Staubli VAL3: Deplacement.pgx

program Deplacement()
begin
  movej(jInit, flange, mNomSpeed)
  movej(jDest, flange, mNomSpeed)
  waitEndMove()

  do
    waitEndMove()
    //movel(pCarre1, flange, mNomSpeed)
    //movel(pCarre2, flange, mNomSpeed)
    movec(pCarre1, pCarre2, flange, mNomSpeed)
    movej(pCarre3, flange, mNomSpeed)
    movej(pCarre4, flange, mNomSpeed)
  until false
end
